FUNCTION_BLOCK EventDrivenCylinder (* Purely Event-Driven function blocks pattern: double-acting cylinder control with zero BOOL data pins *)
  (* Standard: 61499-2; Description: Copyright (c) 2026 Meisterschulen am Ostbahnhof This program and the accompanying materials are made available under the terms of the Eclipse Public License 2.0 which is available at https://www.eclipse.org/legal/epl-2.0/ SPDX-License-Identifier: EPL-2.0 *)
  (* Version 1.0, 2026-08-31, Franz Höpfinger, Meisterschulen am Ostbahnhof, Purely Event-Driven function blocks design pattern (IEC 61499 primer course, Module 6, Valeriy Vyatkin, slide 64). Interface names read directly off the slide's transformed DoubleActingCylinder icon; exact ECC transition wiring is this repo's own consistent reconstruction, not pixel-verified against the compressed slide diagram - see PurelyEventDrivenPattern.md *)
  PACKAGE Meins::DesingPatterns::PurelyEventDrivenPattern;
  (* Documentation:
  Fully event-driven double-acting cylinder controller for the Purely Event-Driven function blocks design pattern (IEC 61499 primer course, Module 6, Valeriy Vyatkin, slide 64) - the transformed end state of the slide's DoubleActingCylinder example.
   Zero BOOL data pins. Position sensors are wired in as events (AT_HOME/AT_END, fired once by the physical sensor edge) instead of continuously-polled BOOL inputs; actuator commands are events (EXTEND/RETRACT) fired directly by the ECC instead of BOOL outputs needing a one-line assignment algorithm. No algorithms at all are needed anywhere in this block - purely event routing.
   Cycle: START → idle at HOME; EXTEND_REQ → fires EXTEND, waits for AT_END → fires STOP+CNF → idle at EXTENDED; RETRACT_REQ → fires RETRACT, waits for AT_HOME → fires STOP+CNF → back to HOME.
   Because there are no data pins, this block is directly testable in FORTE online monitoring - fire the events on the instance by hand, no BOOL values to simulate. See PurelyEventDrivenPattern.md in this folder for the full write-up, including the open question about the exact ECC wiring on the (compressed, hard to pixel-verify) slide diagram.
  *)
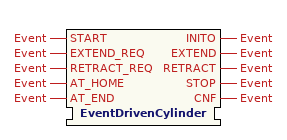
  EVENT_INPUT
    START; (* Initialize: go to the idle HOME state and confirm with INITO *)
    EXTEND_REQ; (* Request the cylinder to extend *)
    RETRACT_REQ; (* Request the cylinder to retract *)
    AT_HOME; (* Fired by the home position sensor: the cylinder is fully retracted *)
    AT_END; (* Fired by the end position sensor: the cylinder is fully extended *)
  END_EVENT
  EVENT_OUTPUT
    INITO; (* Initialization confirmed, now in the idle HOME state *)
    EXTEND; (* Command the actuator to extend *)
    RETRACT; (* Command the actuator to retract *)
    STOP; (* Fired once at the end of every movement (whichever direction), before CNF *)
    CNF; (* Fired once at the end of every movement, confirming the request is complete *)
  END_EVENT
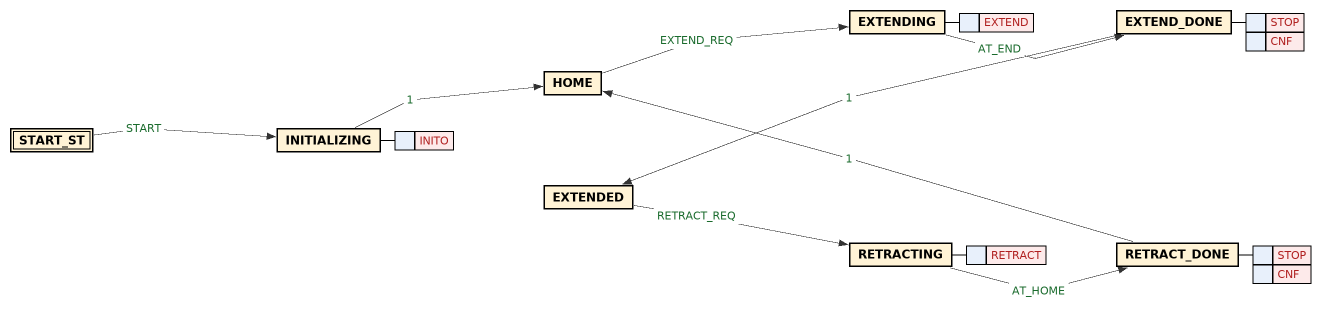
  EC_STATES
    START_ST; (* Uninitialized *)
    INITIALIZING : -> INITO; (* START received: go idle at HOME *)
    HOME; (* Idle, fully retracted *)
    EXTENDING : -> EXTEND; (* Moving out, waiting for AT_END *)
    EXTEND_DONE : -> STOP, -> CNF; (* AT_END received: stop and confirm *)
    EXTENDED; (* Idle, fully extended *)
    RETRACTING : -> RETRACT; (* Moving in, waiting for AT_HOME *)
    RETRACT_DONE : -> STOP, -> CNF; (* AT_HOME received: stop and confirm *)
  END_STATES
  EC_TRANSITIONS
    START_ST TO INITIALIZING := START;
    INITIALIZING TO HOME := 1;
    HOME TO EXTENDING := EXTEND_REQ;
    EXTENDING TO EXTEND_DONE := AT_END;
    EXTEND_DONE TO EXTENDED := 1;
    EXTENDED TO RETRACTING := RETRACT_REQ;
    RETRACTING TO RETRACT_DONE := AT_HOME;
    RETRACT_DONE TO HOME := 1;
  END_TRANSITIONS
END_FUNCTION_BLOCK
